Staubli VAL3: loadEditTraj.pgx

program loadEditTraj(string x_sName)
  local num i
  local num l_nIndex
  local string l_sPath
begin
  // load the traj type
  call saveData:getPathInstr(saveData:sTrajTypeUsing,l_sPath)
  i=trajType:libLoad(l_sPath)
  delay(0)
  if i!=0
    popUpMsg("error load traj type on START "+saveData:sTrajTypeUsing+toString("",i))
  endIf
  // save the name
  sTrajName=x_sName
end
